TYPE ST_JogCommands :
STRUCT
	JogForward   : BOOL;
	JogBackwards : BOOL;
END_STRUCT
END_TYPE

(* stored: Version 1.1.0.1, ProductVersion 3.1.4024.12
   DUT ST_JogCommands: Id {2c9de382-7562-4e56-adee-153efa86e4f5} *)
